FUNCTION_BLOCK PositionMarkerFSA (* AR adapter wrapper around PositionMarkerFS — accepts the Sollwert REAL value via AR adapter socket instead of a plain REQ/rValue pair *)
  (* Standard: ISO 11783-6; Description: Copyright (c) 2026 Meisterschulen am Ostbahnhof This program and the accompanying materials are made available under the terms of the Eclipse Public License 2.0 which is available at https://www.eclipse.org/legal/epl-2.0/ SPDX-License-Identifier: EPL-2.0 Same wrapper shape as Q_NumericValue_PHYSA around Q_NumericValue_PHYS: the AR adapter socket's rPhys value drives the internally-owned PositionMarkerFS instance's REQ/rValue directly. xOver/xUnder are re-exposed as AX adapter plugs, exactly like Q_NumericValue_PHYSA does. *)
  (* Version 1.1, 2026-09-05, Franz Höpfinger, Meisterschulen am Ostbahnhof, Add xScale flag, passed through to the internal PositionMarkerFS *)
  (* Version 1.0, 2026-09-05, Franz Höpfinger, Meisterschulen am Ostbahnhof, initial API and implementation and/or initial documentation *)
  PACKAGE isobus::UT::Q;
  IMPORT isobus::utils::childposition::PositionMarker_S;
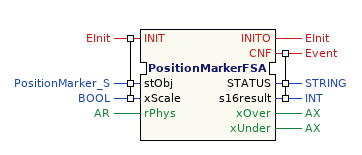
  EVENT_INPUT
    INIT : EInit WITH stObj, xScale; (* Service Initialization *)
  END_EVENT
  EVENT_OUTPUT
    INITO : EInit; (* Initialization Confirm *)
    CNF WITH STATUS, s16result; (* Confirmation of Requested Service *)
  END_EVENT
  VAR_INPUT
    stObj : isobus::utils::childposition::PositionMarker_S; (* Marker object pool properties (child/parent IDs, travel bounds, center offset), snapshotted at INIT *)
    xScale : BOOL := FALSE; (* FALSE (default) = bypass. TRUE = scale by the DM/SKM factor. Passed straight through to the internal PositionMarkerFS instance. *)
  END_VAR
  VAR_OUTPUT
    STATUS : STRING; (* Service Status - passthrough from the internal PositionMarkerFS *)
    s16result : INT; (* retval - passthrough from the internal PositionMarkerFS *)
  END_VAR
  SOCKETS
    rPhys : adapter::types::unidirectional::AR; (* Physical REAL value input *)
  END_SOCKETS
  PLUGS
    xOver : adapter::types::unidirectional::AX; (* rValue (after adding stObj.r32Center) exceeded stObj.r32MaxPos and was clamped *)
    xUnder : adapter::types::unidirectional::AX; (* rValue (after adding stObj.r32Center) fell below stObj.r32MinPos and was clamped *)
  END_PLUGS
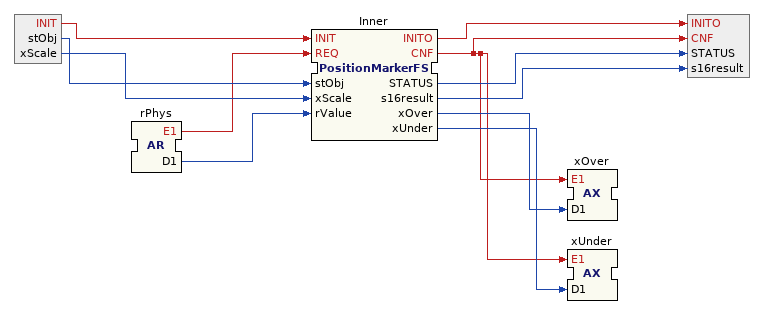
  FBS
    Inner : isobus::UT::Q::PositionMarkerFS;
  END_FBS
  EVENT_CONNECTIONS
    INIT TO Inner.INIT;
    rPhys.E1 TO Inner.REQ;
    Inner.INITO TO INITO;
    Inner.CNF TO CNF;
    Inner.CNF TO xOver.E1;
    Inner.CNF TO xUnder.E1;
  END_CONNECTIONS
  DATA_CONNECTIONS
    stObj TO Inner.stObj;
    xScale TO Inner.xScale;
    rPhys.D1 TO Inner.rValue;
    Inner.STATUS TO STATUS;
    Inner.s16result TO s16result;
    Inner.xOver TO xOver.D1;
    Inner.xUnder TO xUnder.D1;
  END_CONNECTIONS
END_FUNCTION_BLOCK
